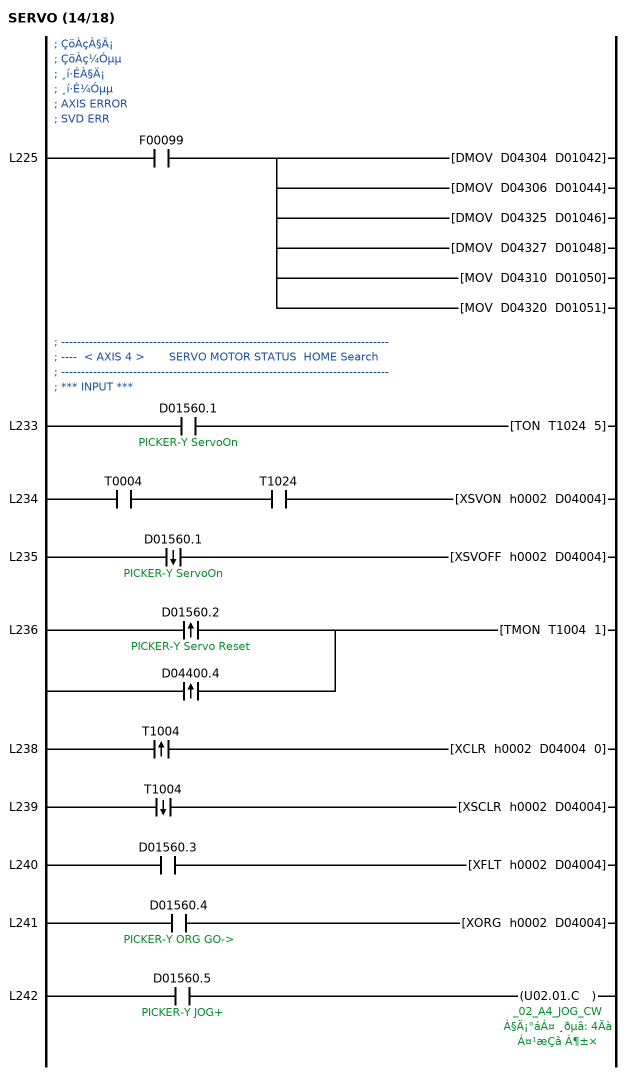
; L225
LOAD      F00099
DMOV      D04304 D01042
DMOV      D04306 D01044
DMOV      D04325 D01046
DMOV      D04327 D01048
MOV       D04310 D01050
MOV       D04320 D01051
// output comment: ÇöÀçÀ§Ä¡
// output comment: ÇöÀç¼Óµµ
// output comment: ¸í·ÉÀ§Ä¡
// output comment: ¸í·É¼Óµµ
// output comment: AXIS ERROR
// output comment: SVD ERR
// ----------------------------------------------------------------------------------
// 
// ----  < AXIS 4 >       SERVO MOTOR STATUS  HOME Search
// 
// ----------------------------------------------------------------------------------
// *** INPUT ***
; L233
LOAD      D01560.1	// PICKER-Y ServoOn
TON       T1024 5
; L234
LOAD      T0004
AND       T1024
XSVON     h0002 D04004
; L235
LOADN     D01560.1	// PICKER-Y ServoOn
XSVOFF    h0002 D04004
; L236
LOADP     D01560.2	// PICKER-Y Servo Reset
ORP       D04400.4
TMON      T1004 1
; L238
LOADP     T1004
XCLR      h0002 D04004 0
; L239
LOADN     T1004
XSCLR     h0002 D04004
; L240
LOAD      D01560.3
XFLT      h0002 D04004
; L241
LOAD      D01560.4	// PICKER-Y ORG GO->
XORG      h0002 D04004
; L242
LOAD      D01560.5	// PICKER-Y JOG+
OUT       U02.01.C	// _02_A4_JOG_CW À§Ä¡°áÁ¤ ¸ðµâ: 4Ãà Á¤¹æÇâ Á¶±×

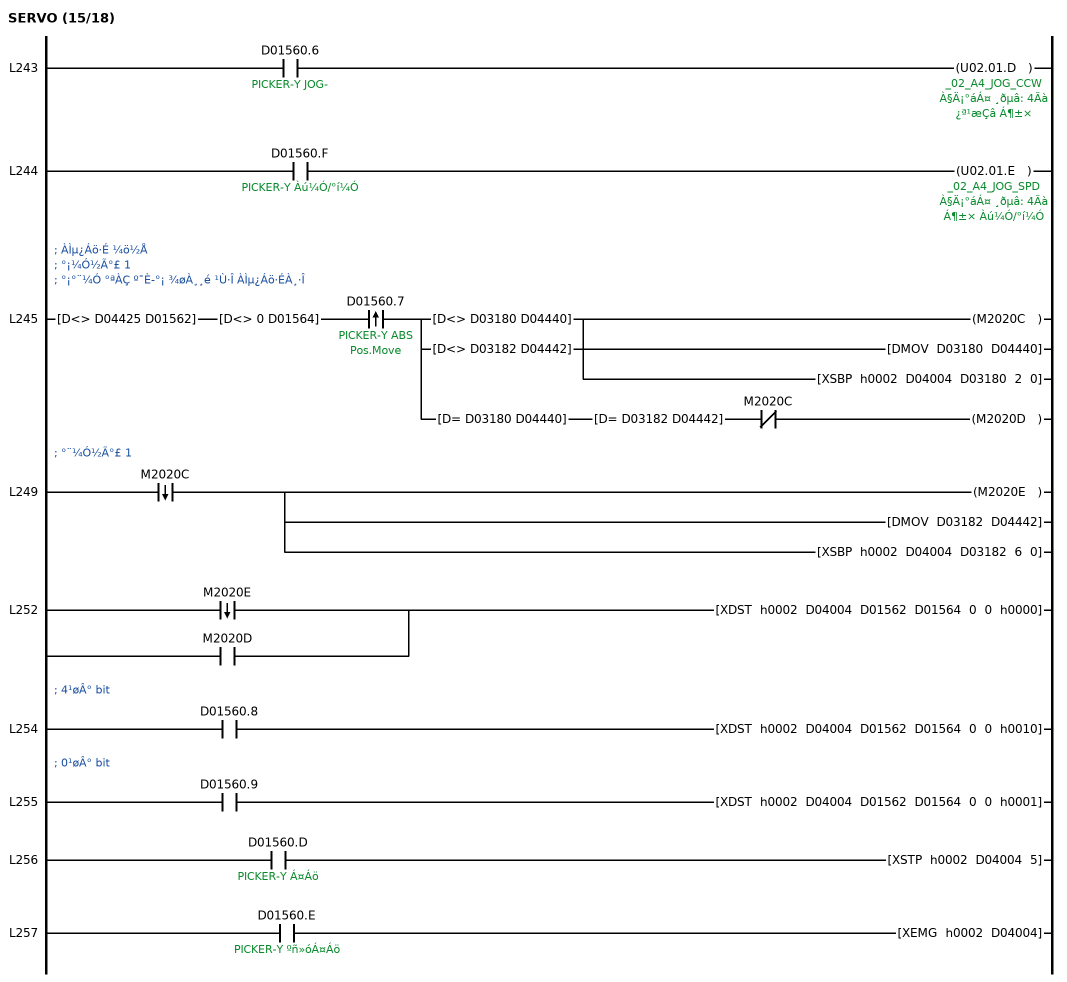
; L243
LOAD      D01560.6	// PICKER-Y JOG-
OUT       U02.01.D	// _02_A4_JOG_CCW À§Ä¡°áÁ¤ ¸ðµâ: 4Ãà ¿ª¹æÇâ Á¶±×
; L244
LOAD      D01560.F	// PICKER-Y Àú¼Ó/°í¼Ó
OUT       U02.01.E	// _02_A4_JOG_SPD À§Ä¡°áÁ¤ ¸ðµâ: 4Ãà Á¶±× Àú¼Ó/°í¼Ó
; L245
LOADD<>   D04425 D01562
ANDD<>    0 D01564
ANDP      D01560.7	// PICKER-Y ABS Pos.Move
MPUSH
LOADD<>   D03180 D04440
ORD<>     D03182 D04442
AND LOAD
OUT       M2020C
DMOV      D03180 D04440
XSBP      h0002 D04004 D03180 2 0
MPOP
ANDD=     D03180 D04440
ANDD=     D03182 D04442
AND NOT   M2020C
OUT       M2020D
// output comment: ÀÌµ¿Áö·É ¼ö½Å
// output comment: °¡¼Ó½Ã°£ 1
// output comment: °¡°¨¼Ó °ªÀÇ º¯È­°¡ ¾øÀ¸¸é ¹Ù·Î ÀÌµ¿Áö·ÉÀ¸·Î
; L249
LOADN     M2020C
OUT       M2020E
DMOV      D03182 D04442
XSBP      h0002 D04004 D03182 6 0
// output comment: °¨¼Ó½Ã°£ 1
; L252
LOADN     M2020E
OR        M2020D
XDST      h0002 D04004 D01562 D01564 0 0 h0000
; L254
LOAD      D01560.8
XDST      h0002 D04004 D01562 D01564 0 0 h0010
// output comment: 4¹øÂ° bit
; L255
LOAD      D01560.9
XDST      h0002 D04004 D01562 D01564 0 0 h0001
// output comment: 0¹øÂ° bit
; L256
LOAD      D01560.D	// PICKER-Y Á¤Áö
XSTP      h0002 D04004 5
; L257
LOAD      D01560.E	// PICKER-Y ºñ»óÁ¤Áö
XEMG      h0002 D04004

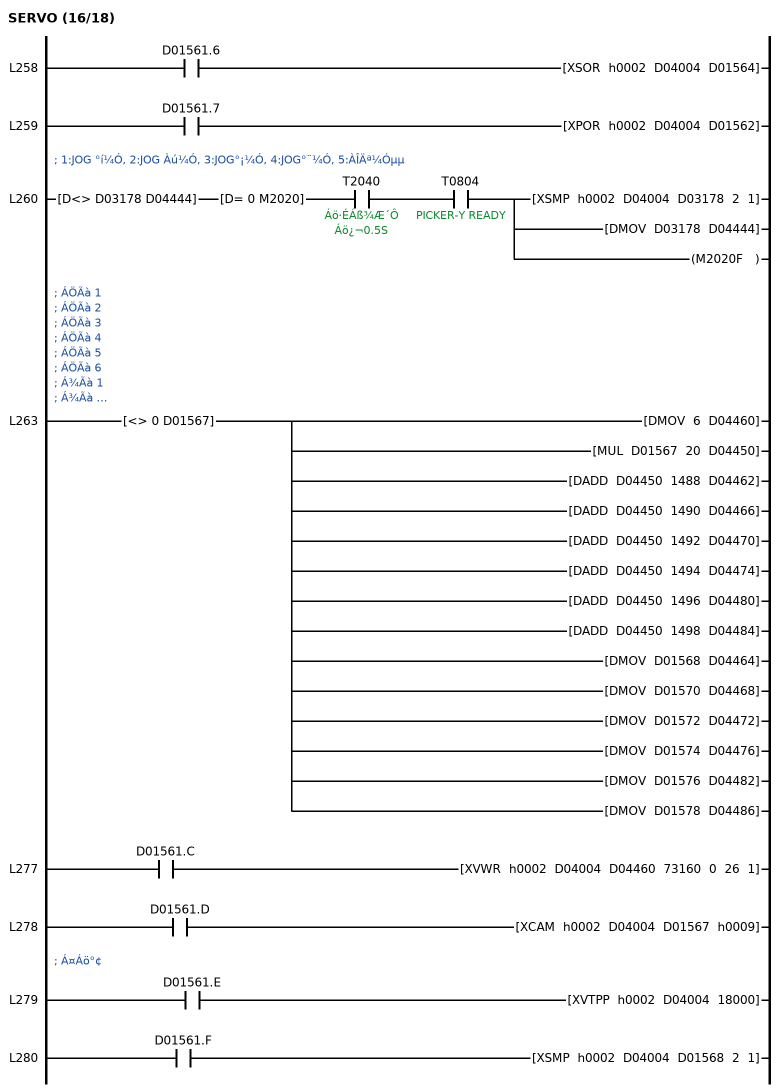
; L258
LOAD      D01561.6
XSOR      h0002 D04004 D01564
; L259
LOAD      D01561.7
XPOR      h0002 D04004 D01562
; L260
LOADD<>   D03178 D04444
ANDD=     0 M2020
AND       T2040	// Áö·ÉÁß¾Æ´Ô Áö¿¬0.5S
AND       T0804	// PICKER-Y READY
XSMP      h0002 D04004 D03178 2 1
DMOV      D03178 D04444
OUT       M2020F
// output comment: 1:JOG °í¼Ó, 2:JOG Àú¼Ó, 3:JOG°¡¼Ó, 4:JOG°¨¼Ó, 5:ÀÎÄª¼Óµµ
; L263
LOAD<>    0 D01567
DMOV      6 D04460
MUL       D01567 20 D04450
DADD      D04450 1488 D04462
DADD      D04450 1490 D04466
DADD      D04450 1492 D04470
DADD      D04450 1494 D04474
DADD      D04450 1496 D04480
DADD      D04450 1498 D04484
DMOV      D01568 D04464
DMOV      D01570 D04468
DMOV      D01572 D04472
DMOV      D01574 D04476
DMOV      D01576 D04482
DMOV      D01578 D04486
// output comment: ÁÖÃà 1
// output comment: ÁÖÃà 2
// output comment: ÁÖÃà 3
// output comment: ÁÖÃà 4
// output comment: ÁÖÃà 5
// output comment: ÁÖÃà 6
// output comment: Á¾Ãà 1
// output comment: Á¾Ãà 2
// output comment: Á¾Ãà 3
// output comment: Á¾Ãà 4
// output comment: Á¾Ãà 5
// output comment: Á¾Ãà 6
; L277
LOAD      D01561.C
XVWR      h0002 D04004 D04460 73160 0 26 1
; L278
LOAD      D01561.D
XCAM      h0002 D04004 D01567 h0009
; L279
LOAD      D01561.E
XVTPP     h0002 D04004 18000
// output comment: Á¤Áö°¢
; L280
LOAD      D01561.F
XSMP      h0002 D04004 D01568 2 1

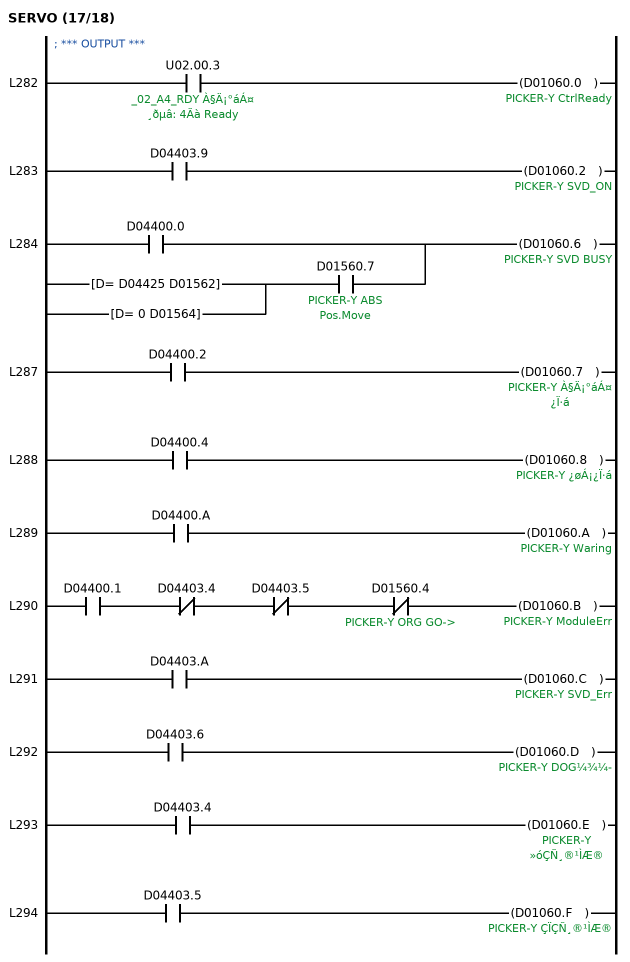
// *** OUTPUT ***
; L282
LOAD      U02.00.3	// _02_A4_RDY À§Ä¡°áÁ¤ ¸ðµâ: 4Ãà Ready
OUT       D01060.0	// PICKER-Y CtrlReady
; L283
LOAD      D04403.9
OUT       D01060.2	// PICKER-Y SVD_ON
; L284
LOAD      D04400.0
LOADD=    D04425 D01562
ORD=      0 D01564
AND       D01560.7	// PICKER-Y ABS Pos.Move
OR LOAD
OUT       D01060.6	// PICKER-Y SVD BUSY
; L287
LOAD      D04400.2
OUT       D01060.7	// PICKER-Y À§Ä¡°áÁ¤ ¿Ï·á
; L288
LOAD      D04400.4
OUT       D01060.8	// PICKER-Y ¿øÁ¡¿Ï·á
; L289
LOAD      D04400.A
OUT       D01060.A	// PICKER-Y Waring
; L290
LOAD      D04400.1
AND NOT   D04403.4
AND NOT   D04403.5
AND NOT   D01560.4	// PICKER-Y ORG GO->
OUT       D01060.B	// PICKER-Y ModuleErr
; L291
LOAD      D04403.A
OUT       D01060.C	// PICKER-Y SVD_Err
; L292
LOAD      D04403.6
OUT       D01060.D	// PICKER-Y DOG¼¾¼­
; L293
LOAD      D04403.4
OUT       D01060.E	// PICKER-Y »óÇÑ¸®¹ÌÆ®
; L294
LOAD      D04403.5
OUT       D01060.F	// PICKER-Y ÇÏÇÑ¸®¹ÌÆ®

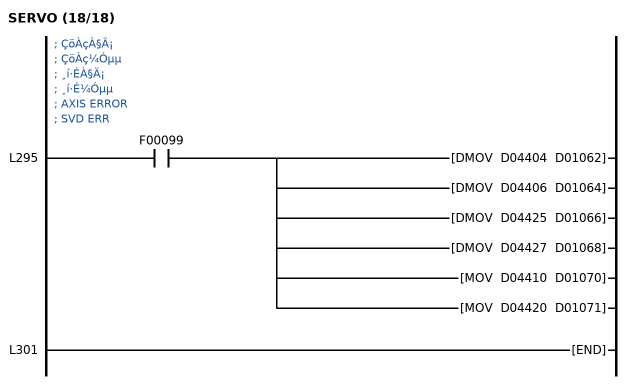
; L295
LOAD      F00099
DMOV      D04404 D01062
DMOV      D04406 D01064
DMOV      D04425 D01066
DMOV      D04427 D01068
MOV       D04410 D01070
MOV       D04420 D01071
// output comment: ÇöÀçÀ§Ä¡
// output comment: ÇöÀç¼Óµµ
// output comment: ¸í·ÉÀ§Ä¡
// output comment: ¸í·É¼Óµµ
// output comment: AXIS ERROR
// output comment: SVD ERR
; L301
END

PROGRAM INTERFACE (task: ½ºÄµ ÇÁ·Î±×·¥)

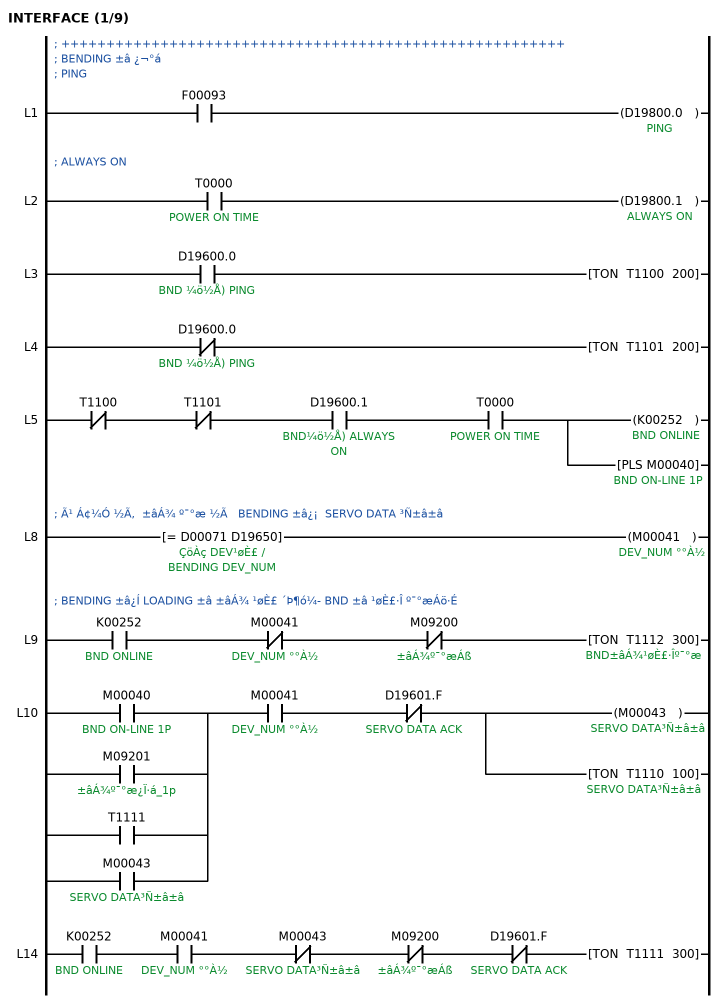
// ++++++++++++++++++++++++++++++++++++++++++++++++++++++++
//    BENDING ±â ¿¬°á
; L1
LOAD      F00093
OUT       D19800.0	// PING
// output comment: PING
; L2
LOAD      T0000	// POWER ON TIME
OUT       D19800.1	// ALWAYS ON
// output comment: ALWAYS ON
; L3
LOAD      D19600.0	// BND ¼ö½Å) PING
TON       T1100 200
; L4
LOAD NOT  D19600.0	// BND ¼ö½Å) PING
TON       T1101 200
; L5
LOAD NOT  T1100
AND NOT   T1101
AND       D19600.1	// BND¼ö½Å) ALWAYS ON
AND       T0000	// POWER ON TIME
OUT       K00252	// BND ONLINE
OUTP      M00040	// BND ON-LINE 1P
// Ã¹ Á¢¼Ó ½Ã,  ±âÁ¾ º¯°æ ½Ã   BENDING ±â¿¡  SERVO DATA ³Ñ±â±â
; L8
LOAD=     D00071 D19650	// ÇöÀç DEV¹øÈ£ / BENDING DEV_NUM
OUT       M00041	// DEV_NUM °°À½
; L9
LOAD      K00252	// BND ONLINE
AND NOT   M00041	// DEV_NUM °°À½
AND NOT   M09200	// ±âÁ¾º¯°æÁß
TON       T1112 300	// BND±âÁ¾¹øÈ£·Îº¯°æ
// output comment: BENDING ±â¿Í LOADING ±â ±âÁ¾ ¹øÈ£ ´Þ¶ó¼­ BND ±â ¹øÈ£·Î º¯°æÁö·É
; L10
LOAD      M00040	// BND ON-LINE 1P
OR        M09201	// ±âÁ¾º¯°æ¿Ï·á_1p
OR        T1111
OR        M00043	// SERVO DATA³Ñ±â±â
AND       M00041	// DEV_NUM °°À½
AND NOT   D19601.F	// SERVO DATA ACK
OUT       M00043	// SERVO DATA³Ñ±â±â
TON       T1110 100	// SERVO DATA³Ñ±â±â
; L14
LOAD      K00252	// BND ONLINE
AND       M00041	// DEV_NUM °°À½
AND NOT   M00043	// SERVO DATA³Ñ±â±â
AND NOT   M09200	// ±âÁ¾º¯°æÁß
AND NOT   D19601.F	// SERVO DATA ACK
TON       T1111 300

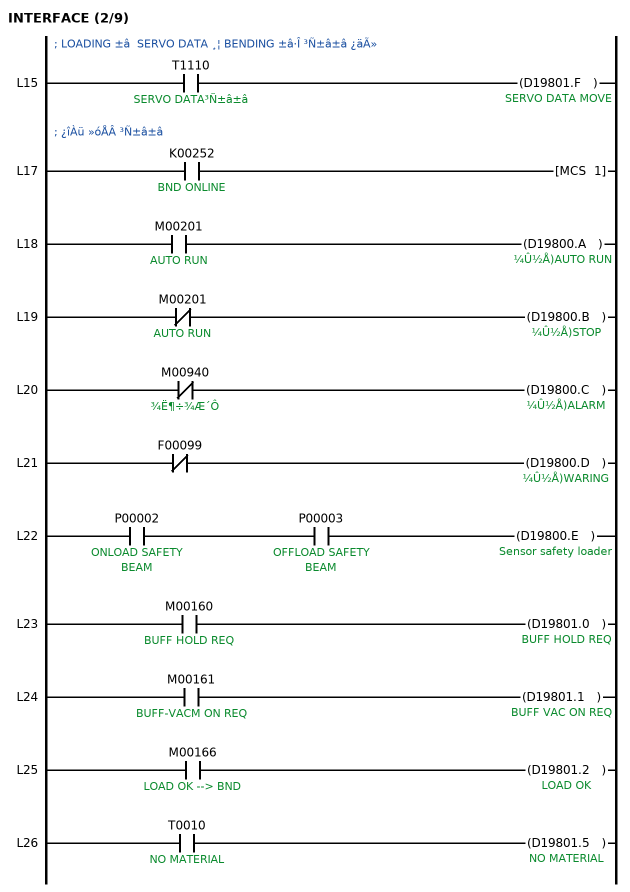
; L15
LOAD      T1110	// SERVO DATA³Ñ±â±â
OUT       D19801.F	// SERVO DATA MOVE
// output comment: LOADING ±â  SERVO DATA ¸¦ BENDING ±â·Î ³Ñ±â±â ¿äÃ»
// ¿îÀü »óÅÂ ³Ñ±â±â
; L17
LOAD      K00252	// BND ONLINE
MCS       1
; L18
LOAD      M00201	// AUTO RUN
OUT       D19800.A	// ¼Û½Å)AUTO RUN
; L19
LOAD NOT  M00201	// AUTO RUN
OUT       D19800.B	// ¼Û½Å)STOP
; L20
LOAD NOT  M00940	// ¾Ë¶÷¾Æ´Ô
OUT       D19800.C	// ¼Û½Å)ALARM
; L21
LOAD NOT  F00099
OUT       D19800.D	// ¼Û½Å)WARING
; L22
LOAD      P00002	// ONLOAD SAFETY BEAM
AND       P00003	// OFFLOAD SAFETY BEAM
OUT       D19800.E	// Sensor safety loader
; L23
LOAD      M00160	// BUFF HOLD REQ
OUT       D19801.0	// BUFF HOLD REQ
; L24
LOAD      M00161	// BUFF-VACM ON REQ
OUT       D19801.1	// BUFF VAC ON REQ
; L25
LOAD      M00166	// LOAD OK --> BND
OUT       D19801.2	// LOAD OK
; L26
LOAD      T0010	// NO MATERIAL
OUT       D19801.5	// NO MATERIAL

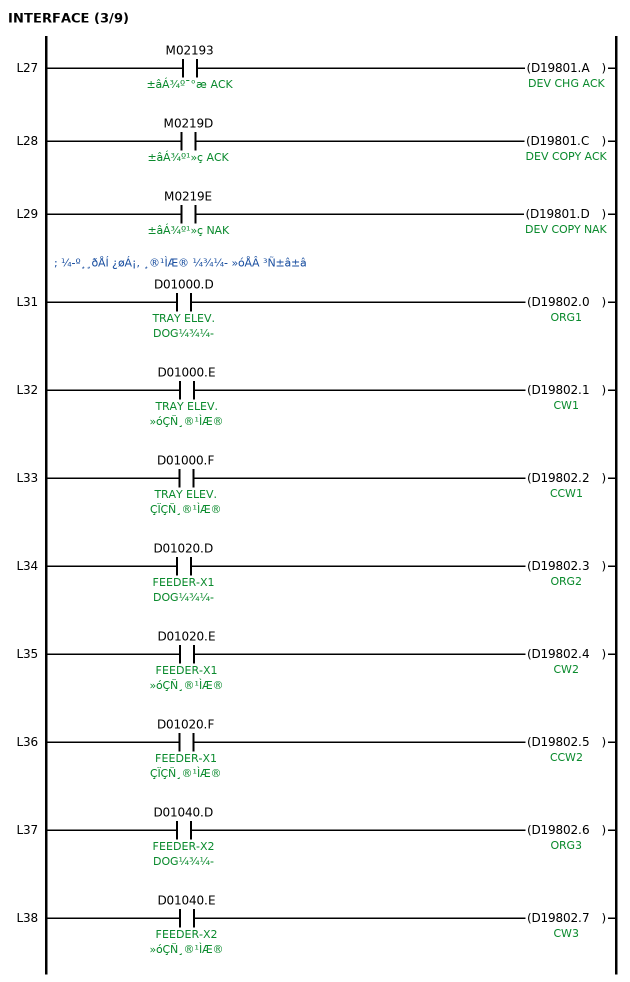
; L27
LOAD      M02193	// ±âÁ¾º¯°æ ACK
OUT       D19801.A	// DEV CHG ACK
; L28
LOAD      M0219D	// ±âÁ¾º¹»ç ACK
OUT       D19801.C	// DEV COPY ACK
; L29
LOAD      M0219E	// ±âÁ¾º¹»ç NAK
OUT       D19801.D	// DEV COPY NAK
// ¼­º¸¸ðÅÍ ¿øÁ¡, ¸®¹ÌÆ® ¼¾¼­ »óÅÂ ³Ñ±â±â
; L31
LOAD      D01000.D	// TRAY ELEV. DOG¼¾¼­
OUT       D19802.0	// ORG1
; L32
LOAD      D01000.E	// TRAY ELEV. »óÇÑ¸®¹ÌÆ®
OUT       D19802.1	// CW1
; L33
LOAD      D01000.F	// TRAY ELEV. ÇÏÇÑ¸®¹ÌÆ®
OUT       D19802.2	// CCW1
; L34
LOAD      D01020.D	// FEEDER-X1 DOG¼¾¼­
OUT       D19802.3	// ORG2
; L35
LOAD      D01020.E	// FEEDER-X1 »óÇÑ¸®¹ÌÆ®
OUT       D19802.4	// CW2
; L36
LOAD      D01020.F	// FEEDER-X1 ÇÏÇÑ¸®¹ÌÆ®
OUT       D19802.5	// CCW2
; L37
LOAD      D01040.D	// FEEDER-X2 DOG¼¾¼­
OUT       D19802.6	// ORG3
; L38
LOAD      D01040.E	// FEEDER-X2 »óÇÑ¸®¹ÌÆ®
OUT       D19802.7	// CW3

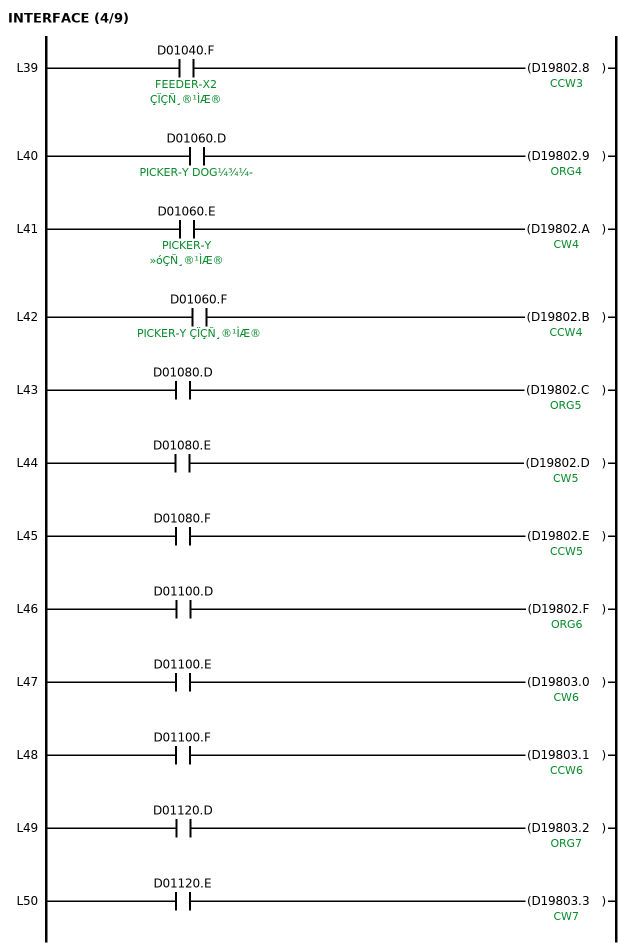
; L39
LOAD      D01040.F	// FEEDER-X2 ÇÏÇÑ¸®¹ÌÆ®
OUT       D19802.8	// CCW3
; L40
LOAD      D01060.D	// PICKER-Y DOG¼¾¼­
OUT       D19802.9	// ORG4
; L41
LOAD      D01060.E	// PICKER-Y »óÇÑ¸®¹ÌÆ®
OUT       D19802.A	// CW4
; L42
LOAD      D01060.F	// PICKER-Y ÇÏÇÑ¸®¹ÌÆ®
OUT       D19802.B	// CCW4
; L43
LOAD      D01080.D
OUT       D19802.C	// ORG5
; L44
LOAD      D01080.E
OUT       D19802.D	// CW5
; L45
LOAD      D01080.F
OUT       D19802.E	// CCW5
; L46
LOAD      D01100.D
OUT       D19802.F	// ORG6
; L47
LOAD      D01100.E
OUT       D19803.0	// CW6
; L48
LOAD      D01100.F
OUT       D19803.1	// CCW6
; L49
LOAD      D01120.D
OUT       D19803.2	// ORG7
; L50
LOAD      D01120.E
OUT       D19803.3	// CW7

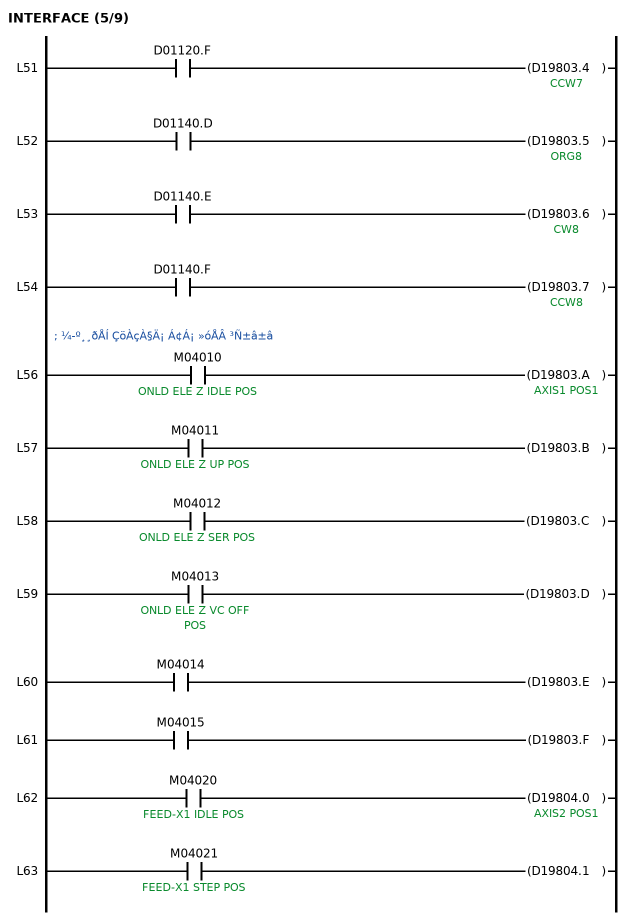
; L51
LOAD      D01120.F
OUT       D19803.4	// CCW7
; L52
LOAD      D01140.D
OUT       D19803.5	// ORG8
; L53
LOAD      D01140.E
OUT       D19803.6	// CW8
; L54
LOAD      D01140.F
OUT       D19803.7	// CCW8
// ¼­º¸¸ðÅÍ ÇöÀçÀ§Ä¡ Á¢Á¡ »óÅÂ ³Ñ±â±â
; L56
LOAD      M04010	// ONLD ELE Z IDLE POS
OUT       D19803.A	// AXIS1 POS1
; L57
LOAD      M04011	// ONLD ELE Z UP POS
OUT       D19803.B
; L58
LOAD      M04012	// ONLD ELE Z SER POS
OUT       D19803.C
; L59
LOAD      M04013	// ONLD ELE Z VC OFF POS
OUT       D19803.D
; L60
LOAD      M04014
OUT       D19803.E
; L61
LOAD      M04015
OUT       D19803.F
; L62
LOAD      M04020	// FEED-X1 IDLE POS
OUT       D19804.0	// AXIS2 POS1
; L63
LOAD      M04021	// FEED-X1 STEP POS
OUT       D19804.1

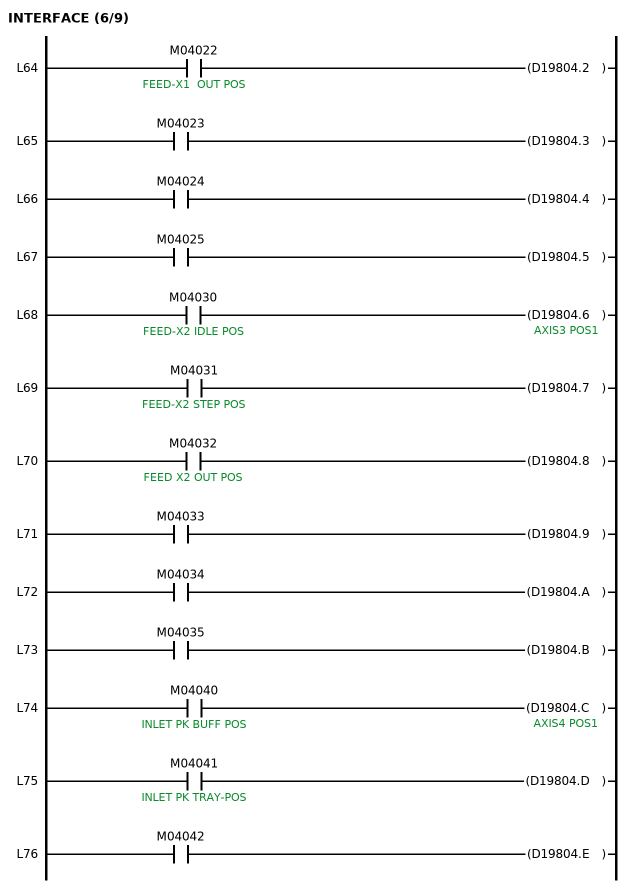
; L64
LOAD      M04022	// FEED-X1  OUT POS
OUT       D19804.2
; L65
LOAD      M04023
OUT       D19804.3
; L66
LOAD      M04024
OUT       D19804.4
; L67
LOAD      M04025
OUT       D19804.5
; L68
LOAD      M04030	// FEED-X2 IDLE POS
OUT       D19804.6	// AXIS3 POS1
; L69
LOAD      M04031	// FEED-X2 STEP POS
OUT       D19804.7
; L70
LOAD      M04032	// FEED X2 OUT POS
OUT       D19804.8
; L71
LOAD      M04033
OUT       D19804.9
; L72
LOAD      M04034
OUT       D19804.A
; L73
LOAD      M04035
OUT       D19804.B
; L74
LOAD      M04040	// INLET PK BUFF POS
OUT       D19804.C	// AXIS4 POS1
; L75
LOAD      M04041	// INLET PK TRAY-POS
OUT       D19804.D
; L76
LOAD      M04042
OUT       D19804.E

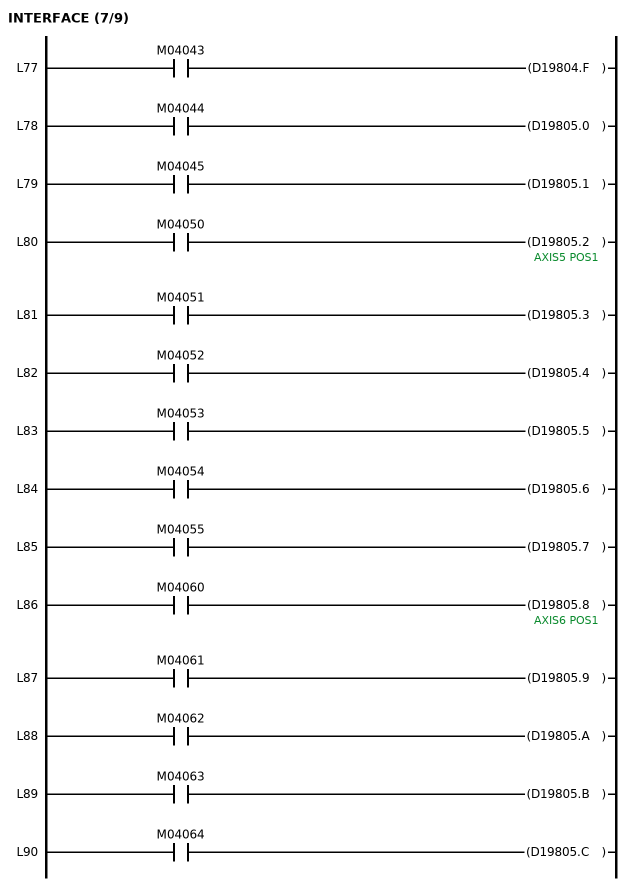
; L77
LOAD      M04043
OUT       D19804.F
; L78
LOAD      M04044
OUT       D19805.0
; L79
LOAD      M04045
OUT       D19805.1
; L80
LOAD      M04050
OUT       D19805.2	// AXIS5 POS1
; L81
LOAD      M04051
OUT       D19805.3
; L82
LOAD      M04052
OUT       D19805.4
; L83
LOAD      M04053
OUT       D19805.5
; L84
LOAD      M04054
OUT       D19805.6
; L85
LOAD      M04055
OUT       D19805.7
; L86
LOAD      M04060
OUT       D19805.8	// AXIS6 POS1
; L87
LOAD      M04061
OUT       D19805.9
; L88
LOAD      M04062
OUT       D19805.A
; L89
LOAD      M04063
OUT       D19805.B
; L90
LOAD      M04064
OUT       D19805.C

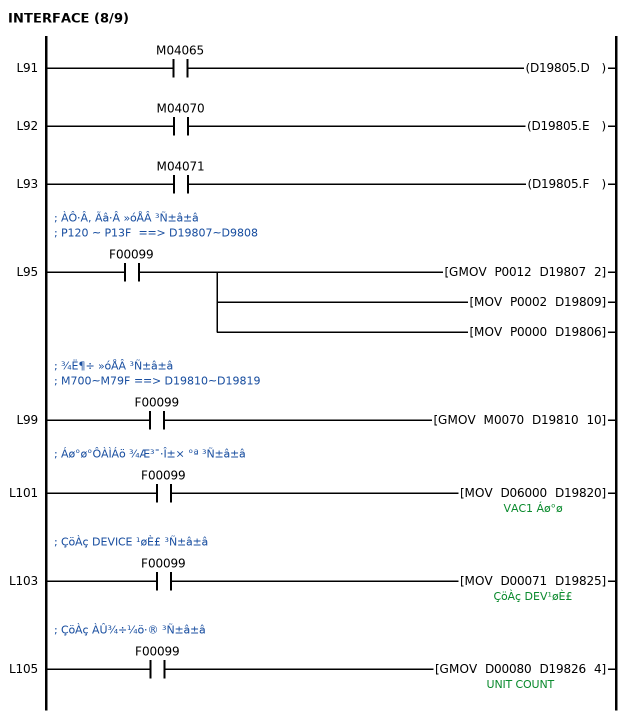
; L91
LOAD      M04065
OUT       D19805.D
; L92
LOAD      M04070
OUT       D19805.E
; L93
LOAD      M04071
OUT       D19805.F
// ÀÔ·Â, Ãâ·Â »óÅÂ ³Ñ±â±â
; L95
LOAD      F00099
GMOV      P0012 D19807 2
MOV       P0002 D19809
MOV       P0000 D19806
// output comment: P120 ~ P13F  ==> D19807~D9808
// ¾Ë¶÷ »óÅÂ ³Ñ±â±â
; L99
LOAD      F00099
GMOV      M0070 D19810 10
// output comment: M700~M79F ==> D19810~D19819
// Áø°ø°ÔÀÌÁö ¾Æ³¯·Î±× °ª ³Ñ±â±â
; L101
LOAD      F00099
MOV       D06000 D19820	// VAC1 Áø°ø
// ÇöÀç DEVICE ¹øÈ£ ³Ñ±â±â
; L103
LOAD      F00099
MOV       D00071 D19825	// ÇöÀç DEV¹øÈ£
// ÇöÀç ÀÛ¾÷¼ö·® ³Ñ±â±â
; L105
LOAD      F00099
GMOV      D00080 D19826 4	// UNIT COUNT

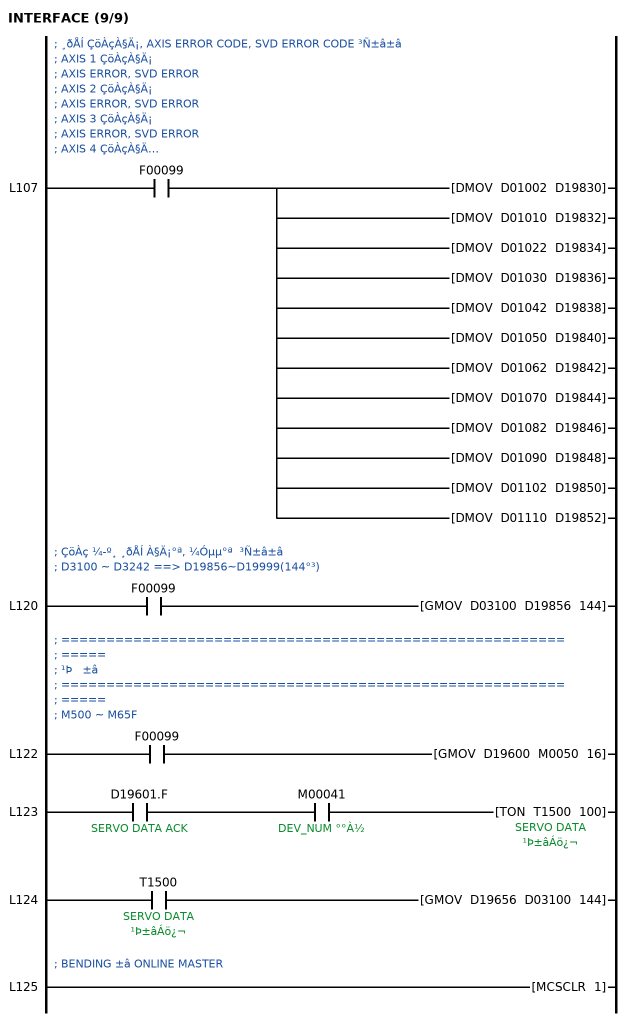
// ¸ðÅÍ ÇöÀçÀ§Ä¡, AXIS ERROR CODE, SVD ERROR CODE ³Ñ±â±â
; L107
LOAD      F00099
DMOV      D01002 D19830
DMOV      D01010 D19832
DMOV      D01022 D19834
DMOV      D01030 D19836
DMOV      D01042 D19838
DMOV      D01050 D19840
DMOV      D01062 D19842
DMOV      D01070 D19844
DMOV      D01082 D19846
DMOV      D01090 D19848
DMOV      D01102 D19850
DMOV      D01110 D19852
// output comment: AXIS 1 ÇöÀçÀ§Ä¡
// output comment: AXIS ERROR, SVD ERROR
// output comment: AXIS 2 ÇöÀçÀ§Ä¡
// output comment: AXIS ERROR, SVD ERROR
// output comment: AXIS 3 ÇöÀçÀ§Ä¡
// output comment: AXIS ERROR, SVD ERROR
// output comment: AXIS 4 ÇöÀçÀ§Ä¡
// output comment: AXIS ERROR, SVD ERROR
// output comment: AXIS 5 ÇöÀçÀ§Ä¡
// output comment: AXIS ERROR, SVD ERROR
// output comment: AXIS 6 ÇöÀçÀ§Ä¡
// output comment: AXIS ERROR, SVD ERROR
// ÇöÀç ¼­º¸ ¸ðÅÍ À§Ä¡°ª, ¼Óµµ°ª  ³Ñ±â±â
; L120
LOAD      F00099
GMOV      D03100 D19856 144
// output comment: D3100 ~ D3242 ==> D19856~D19999(144°³)
// =============================================================
// 
// 
//       ¹Þ   ±â
//       
//       
// =============================================================
; L122
LOAD      F00099
GMOV      D19600 M0050 16
// output comment: M500 ~ M65F
; L123
LOAD      D19601.F	// SERVO DATA ACK
AND       M00041	// DEV_NUM °°À½
TON       T1500 100	// SERVO DATA ¹Þ±âÁö¿¬
; L124
LOAD      T1500	// SERVO DATA ¹Þ±âÁö¿¬
GMOV      D19656 D03100 144
; L125
MCSCLR    1
// output comment: BENDING ±â ONLINE MASTER

VARIABLES AND COMMENTS (devices not used above)
D01000.1	BIT	TRAY ELEV. SVDÁØºñ»óÅÂ
D01000.4	BIT	TRAY ELEV. reset Áö·É¿Ï·á
D01000.9	BIT	TRAY ELEV. StopCommd
D01020.1	BIT	FEEDER-X1 SVDÁØºñ»óÅÂ
D01020.4	BIT	FEEDER-X1 reset Áö·É¿Ï·á
D01020.9	BIT	FEEDER-X1 StopCommd
D01040.1	BIT	FEEDER-X2 SVDÁØºñ»óÅÂ
D01040.4	BIT	FEEDER-X2 reset Áö·É¿Ï·á
D01040.9	BIT	FEEDER-X2 StopCommd
D01060.1	BIT	PICKER-Y SVDÁØºñ»óÅÂ
D01060.4	BIT	PICKER-Y reset Áö·É¿Ï·á
D01060.9	BIT	PICKER-Y StopCommd
P00137	BIT	ONLOAD TRAY SIDE CLAMP CLOSE
M00523	BIT	BND)BUFF VAC ON
M00560	BIT	¼Ó¼Ò¼ÂÆÃ¿ë °­Á¦Ãâ·Â1
M00726	BIT	-
M0078A	BIT	INLET 4th PICKER VACUUM 4 ALARM
M0078B	BIT	INLET 5th PICKER VACUUM 5 ALARM